(* IEC 61131-3 sources: windowtracking/src/Trigger, 6 files *)

(* ---- ITriggerEvent.st ---- *)
USING Simatic.Ax.WindowTracking.Events;

NAMESPACE Simatic.Ax.WindowTracking.VirtualTrigger
    INTERFACE ITriggerEvent
        METHOD Action : EventStatus
            VAR_INPUT
                te : IVirtualTrigger;
                tw : ITransportWindow;
            END_VAR
        END_METHOD
    END_INTERFACE

END_NAMESPACE

(* ---- ITriggerList.st ---- *)
NAMESPACE Simatic.Ax.WindowTracking
    INTERFACE ITriggerList

        METHOD Add : BOOL
            VAR_INPUT
                tp : IVirtualTrigger;
            END_VAR
        END_METHOD

        METHOD Count : UINT
        END_METHOD

        METHOD GetTriggerPoint : IVirtualTrigger
            VAR_INPUT
                Id : UINT;
            END_VAR
        END_METHOD

        METHOD Check : BOOL
             VAR_INPUT
                tw : ITransportWindow;
             END_VAR
        END_METHOD

    END_INTERFACE
END_NAMESPACE

(* ---- IVirtualTrigger.st ---- *)
USING Simatic.Ax.WindowTracking.Events;

NAMESPACE Simatic.Ax.WindowTracking.VirtualTrigger
    INTERFACE IVirtualTrigger

        METHOD ActivateEvent : EventStatus
            VAR_INPUT
                tw : ITransportWindow;
            END_VAR
        END_METHOD

        METHOD IsActivated
        END_METHOD

        METHOD  IsEnabled : BOOL
        END_METHOD

        METHOD GetID : UINT
        END_METHOD

        METHOD GetPosition : DINT
        END_METHOD

    END_INTERFACE
END_NAMESPACE

(* ---- TriggerList.st ---- *)
NAMESPACE Simatic.Ax.WindowTracking.Trigger
    CLASS TriggerList IMPLEMENTS ITriggerList
        VAR PUBLIC
            PositiveTolerace : DINT := 5;
            NegativeTolerance : DINT := 5;
        END_VAR
        VAR PROTECTED
            _triggerPointList : ARRAY[UINT#0..BUF_SIZE - UINT#1] OF IVirtualTrigger;
            _count : UINT;
        END_VAR

        VAR CONSTANT
            BUF_SIZE : UINT := UINT#100;
        END_VAR

        METHOD PUBLIC Add : BOOL
            VAR_INPUT
                tp : IVirtualTrigger;
            END_VAR
            IF (_count < BUF_SIZE) THEN
                _triggerPointList[_count] := tp;
                _count := _count + UINT#1;
            ELSE
                Add := FALSE;
            END_IF;
        END_METHOD

        METHOD PUBLIC Count : UINT
            Count := _count;
        END_METHOD

        METHOD PUBLIC GetTriggerPoint : IVirtualTrigger
            VAR_INPUT
                Id : UINT;
            END_VAR
            VAR_TEMP
                i : UINT;
            END_VAR
            FOR i := UINT#0 TO THIS.Count() - UINT#1 DO
                IF (_triggerPointList[i] = NULL) THEN
                    GetTriggerPoint := NULL;
                    RETURN;
                END_IF;
                IF (_triggerPointList[i].GetId() = Id) THEN
                    GetTriggerPoint := _triggerPointList[i];
                    RETURN;
                END_IF;
            END_FOR;
            GetTriggerPoint := NULL;
        END_METHOD

        METHOD PUBLIC Check : BOOL
            VAR_INPUT
                tw : ITransportWindow;
            END_VAR
            VAR_TEMP
                i : UINT;
                o : IVirtualTrigger;
            END_VAR
            FOR i := UINT#0 TO THIS.Count() - UINT#1 DO
                o := _triggerPointList[i];
                IF (o <> NULL) THEN
                    IF (THIS.InRange(sp := o.GetPosition(), value := tw.GetPosition(), ul := PositiveTolerace, ll := NegativeTolerance)) THEN
                        o.ActivateEvent(tw);
                    END_IF;
                END_IF;
            END_FOR;
        END_METHOD

        METHOD PUBLIC InRange : BOOL
             VAR_INPUT
                sp : DINT;
                value : DINT;
                ul : DINT;
                ll : DINT;
             END_VAR
             VAR_TEMP
                _ul : DINT;
                _ll : DINT;
             END_VAR;
             _ul := sp + ul;
             _ll := sp - ll;

             InRange := value >= _ll AND value <= _ul;
        END_METHOD

    END_CLASS

END_NAMESPACE

(* ---- VirtualTrigger.st ---- *)
USING Simatic.Ax.WindowTracking.EventHandler;
NAMESPACE Simatic.Ax.WindowTracking.Trigger
    CLASS VirtualTrigger IMPLEMENTS IVirtualTrigger

        VAR PUBLIC
            Position : DINT;
            Id : UINT;
            EventHandler : ITriggerEvent;
            PositiveTolerace : DINT := -1;
            NegativeTolerance : DINT := -1;
        END_VAR

        VAR PROTECTED
            _isActiavted : BOOL;
            _activateOld : BOOL;
        END_VAR

        METHOD PUBLIC ActivateEvent : EventStatus
            VAR_INPUT
                tw : ITransportWindow;
            END_VAR

            IF EventHandler <> NULL THEN
                IF THIS.IsEnabled() THEN
                    ActivateEvent := EventHandler.Action(te := THIS, tw := tw);
                    RETURN;
                ELSE
                    ActivateEvent := Eventstatus#NotEnabled;
                    RETURN;
                END_IF;
            ELSE
                ActivateEvent := Eventstatus#NullReference;
            END_IF;

        END_METHOD

        METHOD PUBLIC IsActivated : BOOL
            IsActivated := _isActiavted;
        END_METHOD

        METHOD PUBLIC GetID : UINT
            GetID := Id;
        END_METHOD

        METHOD PUBLIC GetPosition : DINT
            GetPosition := Position;
        END_METHOD

        METHOD PUBLIC IsEnabled : BOOL
            IsEnabled := TRUE;
        END_METHOD

        METHOD PUBLIC Check : BOOL
            VAR_INPUT
                tw : ITransportWindow;
                ll : DINT;
                ul : DINT;
            END_VAR
            VAR_TEMP
                _inRange : BOOL;
                _activateRis : BOOL;
                _ul : DINT;
                _ll : DINT;
            END_VAR
            IF (PositiveTolerace = -1) THEN
                _ul := ul;
            ELSE
                _ul := PositiveTolerace;
            END_IF;
            IF (NegativeTolerance = -1) THEN
                _ll := ll;
            ELSE
                _ll := NegativeTolerance;
            END_IF;
            _inRange := THIS.InRange(sp := Position, value := tw.GetPosition(), ul := _ul, ll := _ll);
            _activateRis := _inRange AND NOT _activateOld;
            _activateOld := _inRange;
            IF (_activateRis) THEN
                _isActiavted := TRUE;
                THIS.ActivateEvent(tw);
            END_IF;
            ;
        END_METHOD

        METHOD PUBLIC InRange : BOOL
            VAR_INPUT
               sp : DINT;
               value : DINT;
               ul : DINT;
               ll : DINT;
            END_VAR
            VAR_TEMP
               _ul : DINT;
               _ll : DINT;
            END_VAR;
            _ul := sp + ul;
            _ll := sp - ll;

            InRange := value >= _ll AND value <= _ul;
       END_METHOD
    END_CLASS
END_NAMESPACE

(* ---- VirtualTriggerList.st ---- *)
NAMESPACE Simatic.Ax.WindowTracking.Trigger
    CLASS VirtualTriggerList IMPLEMENTS ITriggerList
        VAR PUBLIC
            PositiveTolerance : DINT := 5;
            NegativeTolerance : DINT := 5;
            TriggerPointList : REF_TO ARRAY[*] OF IVirtualTrigger;
        END_VAR

        VAR PROTECTED

            _count : UINT;
        END_VAR

        METHOD PUBLIC Add : BOOL
            VAR_INPUT
                tp : IVirtualTrigger;
            END_VAR
            IF (_count < UPPER_BOUND(TriggerPointList^, 1)) THEN
                TriggerPointList^[_count] := tp;
                _count := _count + UINT#1;
            ELSE
                Add := FALSE;
            END_IF;
        END_METHOD

        METHOD PUBLIC Count : UINT
            Count := _count;
        END_METHOD

        METHOD PUBLIC GetTriggerPoint : IVirtualTrigger
            VAR_INPUT
                Id : UINT;
            END_VAR
            VAR_TEMP
                i : UINT;
            END_VAR
            FOR i := UINT#0 TO THIS.Count() - UINT#1 DO
                IF (TriggerPointList^[i] = NULL) THEN
                    GetTriggerPoint := NULL;
                    RETURN;
                END_IF;
                IF (TriggerPointList^[i].GetId() = Id) THEN
                    GetTriggerPoint := TriggerPointList^[i];
                    RETURN;
                END_IF;
            END_FOR;
            GetTriggerPoint := NULL;
        END_METHOD

        METHOD PUBLIC Check : BOOL
            VAR_INPUT
                tw : ITransportWindow;
            END_VAR
            VAR_TEMP
                i : UINT;
                o : IVirtualTrigger;
            END_VAR
            IF (THIS.Count() <= UINT#0) THEN
                Check := FALSE;
                RETURN;
            END_IF;
            FOR i := UINT#0 TO THIS.Count() - UINT#1 DO
                o := TriggerPointList^[i];
                IF (o <> NULL) THEN
                    o.Check(tw := tw, ll := NegativeTolerance, ul := PositiveTolerance);
                END_IF;
            END_FOR;
            Check := TRUE;
        END_METHOD

    END_CLASS

END_NAMESPACE
